{attribute 'pack_mode' := '1'} 
TYPE ST_Beckhoff_EL9110 :
STRUCT
	bPowerOk	AT %Q* : BIT := TRUE;
END_STRUCT
END_TYPE

(* stored: Version 1.1.0.1, ProductVersion 3.1.4024.12
   DUT ST_Beckhoff_EL9110: Id {2c5a4b8d-a3bb-0430-1474-78dc38bbbaa8} *)
